// TwinCAT 3 PLC project Horstman
// ProgramVersion: 3.1.4023.0
// libraries:
//   Tc2_Standard, * (Beckhoff Automation GmbH)
//   Tc2_System, * (Beckhoff Automation GmbH)
//   Tc3_Module, * (Beckhoff Automation GmbH)
// project tree:
//   GVLs/ Global_Variables.TcGVL (not stored)
//   / PlcTask.TcTTO (not stored)
//   POUs/ FB_TcJoy.TcPOU (not stored), MAIN.TcPOU

// ---- POUs/MAIN.TcPOU
PROGRAM MAIN
VAR
END_VAR

.Global_Variables.TcJoy();

IF .Global_Variables.TcJoy.bIsActive THEN
	;
END_IF

END_PROGRAM
